// TIA Portal V20 export
TYPE "LER_typeCommunicationDataS2I"
// stored: Access Published
   STRUCT
      UnitStatus : "LER_typeCommunicationUnitStatus";
      Common : "LER_typeCommonDataInspection";
      UnitHmiData : Array[1..50] of "LER_typeUnitHmiData";
      InterfaceData : "LER_typeCommunicationInterfaceData";
   END_STRUCT;
END_TYPE
